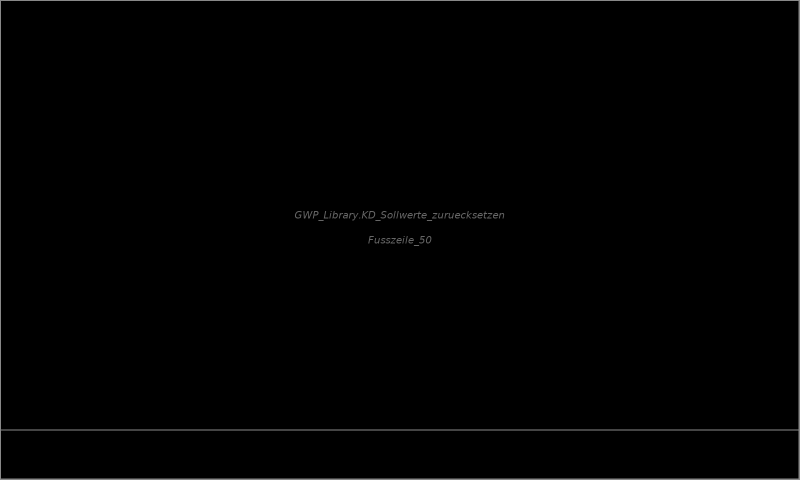
VISUALIZATION KD_Sollwerte_zuruecksetzen  // 800x480
    Frame (0,0 800x430)
        shows GWP_Library.KD_Sollwerte_zuruecksetzen(FB_KD := Main.KD_0)
    Frame (0,0 800x480)
        shows Fusszeile_50()
END_VISUALIZATION

(* stored: Version 1.1.0.1, ProductVersion 3.1.4022.6
   Visu KD_Sollwerte_zuruecksetzen: Id {55e6ffc2-dfc0-46a1-9106-e2f45ea393ad} *)
